// TIA Portal V20 export
TYPE "UDT_Service_Setup"
   STRUCT
      stepOrderOp : UInt;
      stepOrder { ExternalWritable := 'False'} : "UDT_Service_StepOrder";
      parameterIndexOp : UInt;
      parameterIndex { ExternalWritable := 'False'} : Byte;
   END_STRUCT;
END_TYPE
